FUNCTION_BLOCK FB_Medir_SFC
VAR_IN_OUT
    ListadePiezas : ARRAY[1..TAMANO_LISTA_PIEZAS] OF Pieza; 
	TpoMedidor: TIME;
    
END_VAR
VAR_INPUT
    // SFC-Flags
    SFCPause: BOOL;
    SFCReset: BOOL;
    
    // Indicadores de sincronizacion
    Ack: BOOL := TRUE;
    Execute: BOOL;
    
    // Parametros
	NCiclos: INT ;
	AUX_Medidor: INT;
	AUX_FotoElectrico: INT;
	AUX_Metalico: INT;
	
    
    // Entradas
    DetectorInductivo: BOOL;
	DetectorFotoelectrico: BOOL;
	Codificador: UINT;
END_VAR
VAR_OUTPUT
    // Indicadores de sincronizacion
    Done: BOOL;
    Ready: BOOL;
    
    // Salidas
   MedidorBaja: BOOL;
END_VAR
VAR
END_VAR

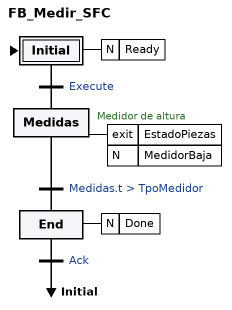
INITIAL_STEP Initial:
    Ready(N);
END_STEP
TRANSITION FROM Initial TO Medidas
    := Execute;
END_TRANSITION
// Medidor de altura
STEP Medidas:
    EstadoPiezas(P0);  // exit action
    MedidorBaja(N);
END_STEP
TRANSITION FROM Medidas TO End
    := Medidas.t > TpoMedidor;
END_TRANSITION
STEP End:
    Done(N);
END_STEP
TRANSITION FROM End TO Initial
    := Ack;
END_TRANSITION

ACTION EstadoPiezas:

//Medidor de altura
AUX_Medidor := AjustarIndice(Nciclos) ;
ListadePiezas[AUX_Medidor].BienColocada := Codificador < 1600; 
ListadePiezas[AUX_Medidor].TipoPieza.Alta := Codificador < 1310;

//Fotoelectrioco
AUX_FotoElectrico := AjustarIndice(Nciclos - 1);
ListadePiezas[AUX_FotoElectrico].TipoPieza.Claro := DetectorFotoelectrico; //TRUE si es clara


//Inductivo
AUX_Metalico := AjustarIndice(Nciclos - 2);
ListadePiezas[AUX_Metalico].TipoPieza.Metalico :=  DetectorInductivo; //TRUE si metalica
END_ACTION

END_FUNCTION_BLOCK

(* stored: Version 1.1.0.1, ProductVersion 3.1.4024.9
   POU FB_Medir_SFC: Id {5b8dfb74-9f25-48a2-a327-170c9156f324}, SpecialFunc None
   Action EstadoPiezas: Id {42a3e1b7-20d3-41fa-877d-84e251584ca8} *)
